INTERFACE I_TcpClient

METHOD M_Connect
VAR_INPUT
	sIP_Address : STRING;
    nPort : UINT;
END_VAR
END_METHOD

METHOD M_Cyclic
VAR_INPUT
END_VAR
END_METHOD

METHOD M_GetData : BOOL;
VAR_INPUT
	pDest : POINTER TO BYTE;
    nSize : UDINT;
END_VAR
END_METHOD

PROPERTY P_HasNewData : bool
GET
END_GET
END_PROPERTY

END_INTERFACE

(* stored: Version 1.1.0.1, ProductVersion 3.1.4024.16
   Itf I_TcpClient: Id {96b47f59-8b05-4a95-ac7f-71e9d8a39dab}
   Method M_Connect: Id {89b798ef-f26f-46a9-a705-2af8a340cdba}
   Method M_Cyclic: Id {f20db6c8-71b5-47e8-b6cd-85de38bb154d}
   Method M_GetData: Id {1e9d0886-8af9-4a37-b9c2-94d3609b3293}
   Property P_HasNewData: Id {26638b89-eed0-4d00-b49e-9837d211b0be}
   Get Get: Id {74657d1f-5bc6-4285-8354-30e8631811e6} *)
